TYPE Str : STRING(255); END_TYPE

(* stored: Version 1.1.0.1
   DUT Str: Id {fc8d502e-75b1-47b9-b2bf-e0576cb15592} *)
